{attribute 'no_explicit_call' := 'no direct call necessary'}
{attribute 'conditionalshow'}
FUNCTION_BLOCK INTERNAL FB_LogBuilder IMPLEMENTS I_LogBuilder
VAR
	sMessage			: T_MaxString;
	eLogLevel			: E_LogLevel;
	sLogger				: T_MaxString := Const.sGlobalLogger;
	fbLogEntry			: FB_LogEntry();
	iLogEntryAdder		: I_LogEntryAdder;
	nIdx				: UINT;
	refScopedContext	: REFERENCE TO ST_ScopedContextStack;
	iContextBuilder		: I_ContextBuilder;
	bStarted			: BOOL;		// TRUE after StartV2 has been called
	bError				: BOOL;
	(* Phase 6 Stage 4: span reference for explicit log-to-trace correlation.
	   Set via WithSpan for logs that should be correlated to a specific span.
	   NULL (default) means no span correlation. *)
	_pSpan				: REFERENCE TO FB_Span;
END_VAR

METHOD PRIVATE _EnsureStarted
IF bStarted OR bError THEN
	RETURN;
END_IF

fbLogEntry.StartV2(
	pLogger			:= ADR(THIS^.sLogger),
	pMessage		:= ADR(THIS^.sMessage),
	eLogLevel		:= eLogLevel,
	nTimeStampPlc	:= 0,
	nTimeStampClock	:= 0
);
bStarted := TRUE;
END_METHOD

METHOD PRIVATE _IsLogLevelActive : BOOL
VAR_INPUT
END_VAR
// Suppress both when the log level is below the configured threshold AND when
// the service is not reachable. Skipping unreachable logs avoids all downstream
// MEMCPY work (message, logger name, args, context) while disconnected.
_IsLogLevelActive := eLogLevel >= Config.eMaxLogLevel
	AND TcOtelInfo.aTaskInfo[Tc2_System.GETCURTASKINDEXEX()].bConnected;
END_METHOD

METHOD INTERNAL Clear : I_LogBuilder
VAR_IN_OUT
	sMessage		: T_MaxString;
END_VAR
VAR_INPUT
	eLogLevel		: E_LogLevel;
	pLogger			: POINTER TO T_MaxString := 0;
END_VAR
Clear := THIS^;
THIS^.eLogLevel := eLogLevel;
IF NOT _IsLogLevelActive() THEN
	RETURN;
END_IF
THIS^.fbLogEntry.Reset();
THIS^.iContextBuilder := 0;
THIS^._pSpan REF= 0;
THIS^.sMessage := sMessage;
IF pLogger <> 0 THEN
	THIS^.sLogger := pLogger^;
ELSE
	THIS^.sLogger := Const.sGlobalLogger;
END_IF
bStarted := FALSE;
bError := FALSE;
END_METHOD

METHOD CreateLog
IF NOT _IsLogLevelActive() THEN
	RETURN;
END_IF

// Ensure header+message+logger are written (in case no args were added)
_EnsureStarted();

// Context comes after args in the wire format
IF __QUERYINTERFACE(PRG_TaskLog.TaskLogger.TaskContext, iLogEntryAdder) THEN
	iLogEntryAdder.AddToLogEntry(E_Scope.eTask, fbLogEntry);
END_IF

refScopedContext REF= PRG_ScopedContextStack.TaskContextStack;
IF refScopedContext.nScopeContextCount > 0 THEN
	FOR nIdx := 0 TO refScopedContext.nScopeContextCount - 1 DO
		IF __QUERYINTERFACE(refScopedContext.aScopedContext[nIdx], iLogEntryAdder) THEN
			iLogEntryAdder.AddToLogEntry(E_Scope.eScoped, fbLogEntry);
		END_IF
	END_FOR
END_IF

IF iContextBuilder <> 0 AND __QUERYINTERFACE(iContextBuilder, iLogEntryAdder) THEN
	iLogEntryAdder.AddToLogEntry(E_Scope.eLogger, fbLogEntry);
END_IF

fbLogEntry.End();
END_METHOD

METHOD WithAnyArg : I_Logger
VAR_INPUT
	stArg	: ANY;
END_VAR
WithAnyArg := THIS^;
IF NOT _IsLogLevelActive() THEN
	RETURN;
END_IF

// Lazy start: write header+message+logger on first arg
_EnsureStarted();

// Write arg directly into LogEntry buffer (v2 format)
fbLogEntry.AddAnyArg(0, stArg);
END_METHOD

METHOD WithContext : I_Logger
VAR_INPUT
	iContextBuilder	: I_ContextBuilder;
END_VAR
WithContext := THIS^;
IF NOT _IsLogLevelActive() THEN
	RETURN;
END_IF
THIS^.iContextBuilder := iContextBuilder;
END_METHOD

METHOD WithLogger : I_WithContext
VAR_INPUT
	sLogger	: T_MaxString;
END_VAR
WithLogger := THIS^;
IF NOT _IsLogLevelActive() THEN
	RETURN;
END_IF
THIS^.sLogger := sLogger;
END_METHOD

(*
:Description: Bind this log entry to a specific FB_Span for explicit
trace context correlation.

When WithSpan is called, the log message will be associated with the span's
trace_id and span_id in the tc-otel backend, creating an explicit link in
the trace timeline.

Call before CreateLog to take effect. Calling after CreateLog has no effect.

Typical usage:

.. code-block:: pascal

    VAR
        spn : FB_Span;
    END_VAR

    F_Log(E_LogLevel.eInfo, 'operation started')
        .WithSpan(spn)
        .CreateLog();
*)
METHOD PUBLIC WithSpan : I_Logger
VAR_IN_OUT
	span : FB_Span;
END_VAR
WithSpan := THIS^;
IF NOT _IsLogLevelActive() THEN
	RETURN;
END_IF

_pSpan REF= span;
END_METHOD

METHOD WithTArg : I_Logger
VAR_INPUT
	stArg	: T_Arg;
END_VAR
WithTArg := THIS^;
IF NOT _IsLogLevelActive() THEN
	RETURN;
END_IF

// Lazy start: write header+message+logger on first arg
_EnsureStarted();

// Write arg directly into LogEntry buffer
fbLogEntry.AddTArg(0, stArg);
END_METHOD

END_FUNCTION_BLOCK

(* stored: Version 1.1.0.1, ProductVersion 3.1.4026.18
   POU FB_LogBuilder: Id {431f68a7-460e-47c3-bd71-217f559bd016}, SpecialFunc None
   Folder Private: Id {4ef16d42-a2ab-482a-a484-f42954a6e403}
   Method _EnsureStarted: Id {e3604386-9c5c-45a7-9663-936eb9ac80ff}
   Method _IsLogLevelActive: Id {ed00c891-12ea-498a-9892-ef7c629ea7f1}
   Method Clear: Id {b4fa87be-fbb6-485f-9775-709e6fc518bf}
   Method CreateLog: Id {23124095-055b-4642-9cec-439e81a94569}
   Method WithAnyArg: Id {8b10c811-cffb-4efb-98e9-827ac612e8d3}
   Method WithContext: Id {7a50707d-ae3e-4603-8990-842a852e28f7}
   Method WithLogger: Id {66d1aa45-8d1b-4222-99f1-0f681c4fd5d5}
   Method WithSpan: Id {e4a59d0f-0a1f-4759-8c0a-1f2d3e4f5a6b}
   Method WithTArg: Id {d3f48c9f-ff2e-465b-bbd7-5053ade8f282} *)
